FUNCTION_BLOCK FB_System
VAR
	plcStart : PLC_Start;
	plcStop : PLC_Stop;
	plcReset : PLC_Reset;
	
	tcRestart : TC_Restart;
	tcConfig : TC_Config;
END_VAR

{attribute 'TcRpcEnable'}
METHOD configTC : BOOL
VAR_INPUT
END_VAR
tcConfig(
	NETID:= , 
	SET:= TRUE, 
	TMOUT:= , 
	BUSY=> , 
	ERR=> , 
	ERRID=> );
	
tcConfig(
	NETID:= , 
	SET:= FALSE, 
	TMOUT:= , 
	BUSY=> , 
	ERR=> , 
	ERRID=> );
END_METHOD

{attribute 'TcRpcEnable'}
METHOD resetPLC : BOOL
VAR_INPUT
END_VAR
plcReset(
	NETID:= , 
	PORT:= 851, 
	RESET:= TRUE, 
	TMOUT:= , 
	BUSY=> , 
	ERR=> , 
	ERRID=> );
	
plcReset(
	NETID:= , 
	PORT:= 851, 
	RESET:= FALSE, 
	TMOUT:= , 
	BUSY=> , 
	ERR=> , 
	ERRID=> );
END_METHOD

{attribute 'TcRpcEnable'}
METHOD restartTC : BOOL
tcRestart(
	NETID:= , 
	RESTART:= TRUE, 
	TMOUT:= , 
	BUSY=> , 
	ERR=> , 
	ERRID=> );
	
tcRestart(
	NETID:= , 
	RESTART:= FALSE, 
	TMOUT:= , 
	BUSY=> , 
	ERR=> , 
	ERRID=> );
END_METHOD

{attribute 'TcRpcEnable'}
METHOD startPLC : BOOL
plcStart(
	NETID:= '', 
	PORT:= 851, 
	START:= TRUE, 
	TMOUT:= , 
	BUSY=> , 
	ERR=> , 
	ERRID=> );
	
plcStart(
	NETID:= '', 
	PORT:= 851, 
	START:= FALSE, 
	TMOUT:= , 
	BUSY=> , 
	ERR=> , 
	ERRID=> );
END_METHOD

{attribute 'TcRpcEnable'}
METHOD stopPLC : BOOL
plcStop(
	NETID:= '', 
	PORT:= 851, 
	STOP:= TRUE, 
	TMOUT:= , 
	BUSY=> , 
	ERR=> , 
	ERRID=> );
	
plcStop(
	NETID:= '', 
	PORT:= 851, 
	STOP:= FALSE, 
	TMOUT:= , 
	BUSY=> , 
	ERR=> , 
	ERRID=> );
END_METHOD

END_FUNCTION_BLOCK

(* stored: Version 1.1.0.1, ProductVersion 3.1.4024.11
   POU FB_System: Id {3df11356-d723-40c5-bd16-325ffd1c8434}, SpecialFunc None
   Method configTC: Id {10f65ef4-9bbd-4708-becc-480ebe0fe5f3}
   Method resetPLC: Id {4a428e1a-7da5-40b0-b115-7e45ad1d899a}
   Method restartTC: Id {f0606f07-75fa-4988-a608-8d72982073d8}
   Method startPLC: Id {f1e1dfb1-a05a-46a8-95e0-a372db58dbfb}
   Method stopPLC: Id {d85e402a-5466-4cae-a47b-6151c6e3078c} *)
